TEXTLIST AxesMuUnitsTextList
  0 = 'arcsec / year'
  1 = 'mas / year'
  2 = 'deg / year'
  3 = 'rad / year'
   = ''
END_TEXTLIST

(* stored: Version 1.1.0.1, ProductVersion 3.1.4018.5
   TextList AxesMuUnitsTextList: Id {f1fd65f5-b4f8-46f5-80f9-955705eb053d} *)
